(* PLC project SafeLOGIC-1, BrAutomation SafeDESIGNER  4.4.0.0 *)
(* stored: companyURL http://www.br-automation.com, creationDateTime Mon May 10 15:16:52 2021 *)

PROGRAM Main
  VAR  (* added by the conversion: wires and edge detectors of the diagram *)
    _OR_S23_OUT : ANY;
    _SAFEBOOL_TO_BOOL42_OUT : BOOL;
  END_VAR

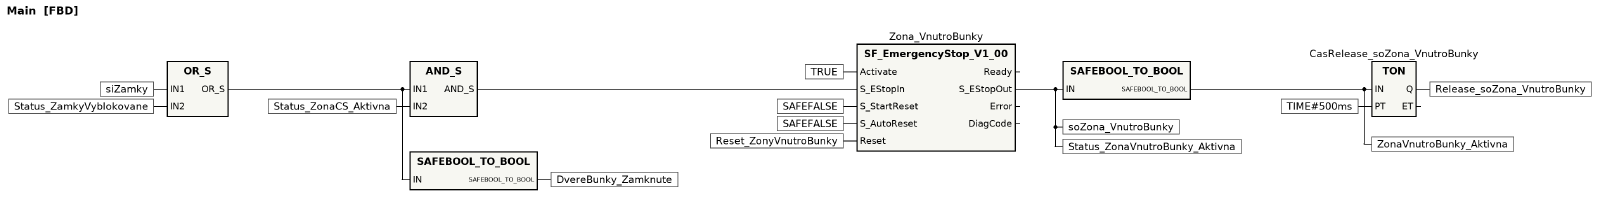
(* FBD diagram, written out as Structured Text *)
_OR_S23_OUT := OR_S(siZamky, Status_ZamkyVyblokovane);
Zona_VnutroBunky(Activate := TRUE, S_EStopIn := AND_S(_OR_S23_OUT, Status_ZonaCS_Aktivna), S_StartReset := SAFEFALSE, S_AutoReset := SAFEFALSE, Reset := Reset_ZonyVnutroBunky);
soZona_VnutroBunky := Zona_VnutroBunky.S_EStopOut;
DvereBunky_Zamknute := SAFEBOOL_TO_BOOL(_OR_S23_OUT);
Status_ZonaVnutroBunky_Aktivna := Zona_VnutroBunky.S_EStopOut;
_SAFEBOOL_TO_BOOL42_OUT := SAFEBOOL_TO_BOOL(Zona_VnutroBunky.S_EStopOut);
CasRelease_soZona_VnutroBunky(IN := _SAFEBOOL_TO_BOOL42_OUT, PT := TIME#500ms);
Release_soZona_VnutroBunky := CasRelease_soZona_VnutroBunky.Q;
ZonaVnutroBunky_Aktivna := _SAFEBOOL_TO_BOOL42_OUT;
END_PROGRAM
